// TIA Portal project "Project8" (V13)
// PDE3422 - Industrial Automation and Control (2017/2018 Assessment)

(* hardware
DEVICE "S7-1200 station_1"  S7-1200 Station
   slot 0: "Rack_0"  Rack  V1.0
   slot 1: "PLC_1"  CPU 1214C DC/DC/DC  6ES7 214-1AG40-0XB0  V4.1
      slot 3: "AQ 1x12BIT_1"  6ES7 232-4HA30-0XB0  V1.0
   slot 2: "DI 8/DQ 8x24VDC_1"  6ES7 223-1BH32-0XB0  V2.0
DEVICE "HMI_1"  KTP700 Basic PN
   slot 0: "HMI"  HMI  6AV2 123-2GB03-0AX0  13.0.1.0
   slot 1: "HMI_RT_1"  KTP700 Basic PN  6AV2 123-2GB03-0AX0  13.0.1.0
   slot 5: "HMI_1.IE_CP_1"  PROFINET Interface
      slot 1: "PROFINET Interface_1"  PROFINET Interface
         slot 1: "Port_1"  Port
*)

// ===== PLC "PLC_1"  CPU 1214C DC/DC/DC =====

VAR_GLOBAL   // PLC tag table "Default tag table"
   "A_IS_EXTENDED" AT %I0.0 : Bool;
   "A_IS_NOT_EXTENDED" AT %I0.1 : Bool;
   "B_IS_EXTENDED" AT %I0.2 : Bool;
   "B_IS_NOT_EXTENDED" AT %I0.3 : Bool;
   "V_IS_EXTENDED" AT %M0.0 : Bool;
   "V_IS_NOT_EXTENDED" AT %M0.1 : Bool;
   "EXTEND_A" AT %Q0.0 : Bool;
   "EXTEND_B" AT %Q0.1 : Bool;
   "EXTEND_V" AT %M0.2 : Bool;
   "PISTON_A_POSITION" AT %MW20 : Int;
   "PISTON_B_POSITION" AT %MW22 : Int;
   "PISTON_V_POSITION" AT %MW24 : Int;
   "N" AT %MW26 : Int;
   "N_MINUS_ONE" AT %MW28 : Int;
   "START_FLAG" AT %M0.3 : Bool;
   "PAUSE_FLAG" AT %M0.4 : Bool;
   "INPUT_VOLTAGE" AT %IW64 : Word;
   "ANALOG_VOLTAGE" AT %MW30 : Int;
   "TEMP_VAR" AT %MD50 : Real;
END_VAR

DATA_BLOCK "MAIN_DATA_BLOCK"   // DB1
{ S7_Optimized_Access := 'FALSE' }
VERSION : 0.1
   VAR
      N : Int;
      TIMER_VALUE_TS : Time;
   END_VAR
BEGIN
END_DATA_BLOCK

DATA_BLOCK "MAIN_ROUNTINE_DB"   // DB2
{ S7_Optimized_Access := 'FALSE' }
VERSION : 0.1
// stored: InstanceOfName MAIN_ROUNTINE
"MAIN_ROUNTINE"
BEGIN
END_DATA_BLOCK

// folder: System blocks/Program resources

DATA_BLOCK "TIMER_11"   // DB4
{ S7_Optimized_Access := 'FALSE' }
AUTHOR : Simatic
FAMILY : IEC
NAME : IEC_TMR
VERSION : 1.0
// stored: InstanceOfName ?
"?"
BEGIN
END_DATA_BLOCK

// folder: (top level)

FUNCTION_BLOCK "MAIN_ROUNTINE"   // FB1, SCL
{ S7_Optimized_Access := 'FALSE' }
VERSION : 0.1
BEGIN
   IF "START_FLAG" = FALSE THEN
       RESET_TIMER(#TIMER_1);
       #COUNT_VAR_1 := 0;
       #"STEP" := 0;
   ELSE
       CASE #"STEP" OF
           0:
               RESET_TIMER(#TIMER_1);
               #COUNT_VAR_1 := 0;

               "EXTEND_A" := TRUE;
               "EXTEND_B" := FALSE;
               #"STEP" := 1;
           1:
               IF "A_IS_EXTENDED" AND "B_IS_NOT_EXTENDED" THEN
                   #TIMER_1(IN := TRUE,
                            PT := #TIMER_1_TIME);
                   #"STEP" := 111;
               END_IF;

           111:
               IF #TIMER_1.Q THEN
                   RESET_TIMER(#TIMER_1);
                   #"STEP" := 2;
               END_IF;

           2:
               "EXTEND_A" := FALSE;
               "EXTEND_B" := TRUE;
               #"STEP" := 3;
           3:
               IF "A_IS_NOT_EXTENDED" AND "B_IS_EXTENDED" THEN
                   #"STEP" := 4;
               END_IF;

           4:
               "EXTEND_B" := FALSE;
               #"STEP" := 5;

           5:
               IF "B_IS_NOT_EXTENDED" THEN
                   #"STEP" := 6;
                   #COUNT_VAR_1 := 0;
               END_IF;

           6:
               IF #COUNT_VAR_1 >= "MAIN_DATA_BLOCK".N THEN
                   #COUNT_VAR_1 := 0;
                   #"STEP" := 10;
               ELSE
                   "EXTEND_A" := TRUE;
                   "EXTEND_V" := TRUE;

                   #"STEP" := 7;
               END_IF;

           7:
               IF "A_IS_EXTENDED" AND "V_IS_EXTENDED" THEN
                   #TIMER_1(IN := TRUE,
                            PT := INT_TO_TIME("ANALOG_VOLTAGE" * 1000));
                   #"STEP" := 8;
               END_IF;

           8:
               IF #TIMER_1.Q THEN
                   RESET_TIMER(#TIMER_1);
                   #"STEP" := 9;
               END_IF;

           9:
               "EXTEND_A" := FALSE;
               "EXTEND_V" := FALSE;

               #"STEP" := 222;

           222:
               IF "A_IS_NOT_EXTENDED" AND "V_IS_NOT_EXTENDED" THEN
                   #"STEP" := 333;
               END_IF;

           333:
               #COUNT_VAR_1 := #COUNT_VAR_1 + 1;

               IF #COUNT_VAR_1 < "MAIN_DATA_BLOCK".N THEN
                   #"STEP" := 6;
               ELSE
                   #COUNT_VAR_1 := 0;
                   #"STEP" := 10;
               END_IF;

           10:
               "EXTEND_V" := TRUE;
               #"STEP" := 11;

           11:
               IF "V_IS_EXTENDED" THEN
                   #TIMER_1(IN := TRUE,
                            PT := #TIMER_1_TIME);
                   #"STEP" := 12;
               END_IF;

           12:
               IF #TIMER_1.Q THEN
                   RESET_TIMER(#TIMER_1);
                   #"STEP" := 13;
               END_IF;

           13:
               "EXTEND_A" := TRUE;
               #"STEP" := 14;

           14:
               IF "A_IS_EXTENDED" THEN
                   #"STEP" := 15;
               END_IF;

           15:
               IF #COUNT_VAR_1 < "N_MINUS_ONE" THEN
                   "EXTEND_V" := FALSE;
                   "EXTEND_A" := FALSE;
                   #"STEP" := 16;
               ELSE
                   #COUNT_VAR_1 := 0;
                   #"STEP" := 21;
               END_IF;

           16:
               IF "V_IS_NOT_EXTENDED" AND "A_IS_NOT_EXTENDED" THEN
                   #TIMER_1(IN := TRUE,
                            PT := INT_TO_TIME("ANALOG_VOLTAGE" * 1000));
                   #"STEP" := 17;
               END_IF;

           17:
               IF #TIMER_1.Q THEN
                   RESET_TIMER(#TIMER_1);
                   #"STEP" := 18;
               END_IF;

           18:
               "EXTEND_V" := TRUE;
               "EXTEND_A" := TRUE;

               #"STEP" := 19;

           19:
               IF "V_IS_EXTENDED" AND "A_IS_EXTENDED" THEN
                   #"STEP" := 20;
               END_IF;

           20:
               #COUNT_VAR_1 := #COUNT_VAR_1 + 1;

               IF #COUNT_VAR_1 < "N_MINUS_ONE" THEN
                   #"STEP" := 15;
               ELSE
                   #COUNT_VAR_1 := 0;
                   #"STEP" := 21;
               END_IF;

           21:
               "EXTEND_V" := FALSE;
               "EXTEND_A" := FALSE;
               "EXTEND_B" := TRUE;

               #"STEP" := 22;

           22:
               IF "V_IS_NOT_EXTENDED" AND "A_IS_NOT_EXTENDED" AND "B_IS_EXTENDED" THEN
                   #"STEP" := 0;
               END_IF;


           23:
               #"STEP" := 0;

       END_CASE;
   END_IF;
END_FUNCTION_BLOCK

ORGANIZATION_BLOCK "Main"   // OB1, LAD, ProgramCycle
TITLE = "Main Program Sweep (Cycle)"
{ S7_Optimized_Access := 'FALSE' }
VERSION : 0.1
BEGIN

REGION Network 1
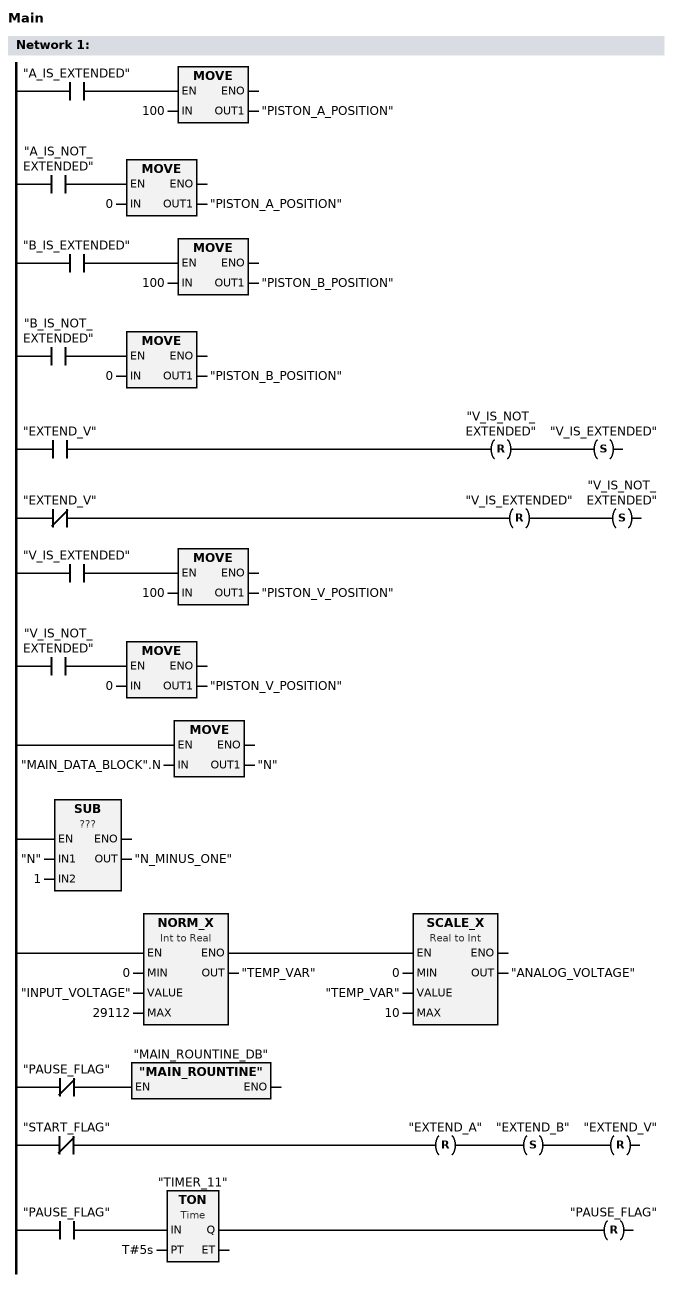
   IF "A_IS_EXTENDED" THEN "PISTON_A_POSITION" := 100; END_IF;
   IF "A_IS_NOT_EXTENDED" THEN "PISTON_A_POSITION" := 0; END_IF;
   IF "B_IS_EXTENDED" THEN "PISTON_B_POSITION" := 100; END_IF;
   IF "B_IS_NOT_EXTENDED" THEN "PISTON_B_POSITION" := 0; END_IF;
   IF "EXTEND_V" THEN
       "V_IS_NOT_EXTENDED" := FALSE;
       "V_IS_EXTENDED" := TRUE;
   END_IF;
   IF NOT "EXTEND_V" THEN
       "V_IS_EXTENDED" := FALSE;
       "V_IS_NOT_EXTENDED" := TRUE;
   END_IF;
   IF "V_IS_EXTENDED" THEN "PISTON_V_POSITION" := 100; END_IF;
   IF "V_IS_NOT_EXTENDED" THEN "PISTON_V_POSITION" := 0; END_IF;
   "N" := "MAIN_DATA_BLOCK".N;
   "N_MINUS_ONE" := "N" - 1;
   "TEMP_VAR" := NORM_X(MIN := 0, VALUE := "INPUT_VOLTAGE", MAX := 29112);
   "ANALOG_VOLTAGE" := SCALE_X(MIN := 0, VALUE := "TEMP_VAR", MAX := 10);
   IF NOT "PAUSE_FLAG" THEN
       "MAIN_ROUNTINE_DB"();   // "MAIN_ROUNTINE"
   END_IF;
   IF NOT "START_FLAG" THEN
       "EXTEND_A" := FALSE;
       "EXTEND_B" := TRUE;
       "EXTEND_V" := FALSE;
   END_IF;
   "TIMER_11".TON(IN := "PAUSE_FLAG", PT := T#5s);
   IF "TIMER_11".Q THEN "PAUSE_FLAG" := FALSE; END_IF;
END_REGION
END_ORGANIZATION_BLOCK

(* ===== HMI "HMI_RT_1" =====
connection "HMI_Connection_1": ETHERNET, SMART_S7_1200_OMS

HMI tags "Default tag table"
   "PISTON_A_POSITION" : Int = PLC "PISTON_A_POSITION", 100 ms
   "PISTON_V_POSITION" : Int = PLC "PISTON_V_POSITION", 100 ms
   "PISTON_B_POSITION" : Int = PLC "PISTON_B_POSITION", 100 ms
   "DATA_BLOCK_N_N" : Int, 100 ms
   "N_MINUS_ONE" : Int = PLC "N_MINUS_ONE", 100 ms
   "START_FLAG" : Bool = PLC "START_FLAG", 100 ms
   "PAUSE_FLAG" : Bool = PLC "PAUSE_FLAG", 100 ms
   "ANALOG_VOLTAGE" : Int = PLC "ANALOG_VOLTAGE", 100 ms

text list "foo": 1 ''; 1 ''; 2 ''; 3 ''

screen "Root screen" 800x480, template "Template_1"
   Button "Button_1" at 247,408 size 179x59
   Button "Button_2" at 247,343 size 179x59
   Button "Button_3" at 433,344 size 120x122
   IOField "I/O field_1" at 688,108 size 96x49
   SymbolicIOField "Symbolic I/O field_1" at 688,210 size 96x52
   TextField "Text field_1" at 712,187 size 72x23
   TextField "Text field_2" at 700,85 size 84x23
   Group "Group" at 68,100 size 139x33
   Group "Group_1" at 68,170 size 139x33
   Group "Group_2" at 68,240 size 139x33
   TextField "Text field_3" at 21,98 size 25x39
   TextField "Text field_4" at 21,170 size 25x39
   TextField "Text field_5" at 21,240 size 25x39
*)